# EPICS substitutions: fastFeedbackApp/Db/iocs/fbckFB02.substitutions
# File fbckFB02.substitutions
#
#
# NOTE - feedback names cannot have any spaces in them
#
# Feedback Types :
#
# define all loops here
file ../../../../db/fbckLoop.db {
  pattern { AR,  LP   ,  LN          }
          { FB02, "TR01"  , "LaunchLoop1"   }
          { FB02, "TR02"  , "LaunchLoop2"   }
          { FB02, "TR03"  , "LaunchLoop3"   }
          { FB02, "TR04"  , "LaunchLoop4"   }
          { FB02, "TR05"  , "LaunchLoop5"   }
# Every IOC will have two spares for on the fly general loop configurations
          { FB02, "GN01"  , "General1"       }
          { FB02, "GN02"  , "General2"       }
# Every IOC will have one longitudinal loop configuration
          { FB02, "LG01"  , "Longitudinal"   }
}
file ../../../../db/fbckIoc.db {
  pattern { AR }
          { FB02 }
}
